TYPE "DecoilersHRot_Manager"
VERSION : 0.1
// Block: DecoilersHRot_Manager
   STRUCT
      EnableStopDoorOpeningReq : Bool;
      EnableStopInPhase : Bool;
      EnableStopProgrammed : Bool;
      Control_ON : Bool;
      Decoiler1_MoveInLine : Bool;
      Decoiler2_MoveInLine : Bool;
      ChangeDecoilerEnable : Bool;
   END_STRUCT;

END_TYPE
